FUNCTION_BLOCK FB_UAnodeReleaseHandleMock_Success IMPLEMENTS I_OPCUA_NodeReleaseHandle
VAR_INPUT
END_VAR
VAR_OUTPUT
END_VAR
VAR
END_VAR

{warning 'add method implementation '}
METHOD start : BOOL
VAR_INPUT
    Execute       : BOOL;
    ConnectionHdl : DWORD;
    NodeHdl       : DWORD;
    Timeout       : TIME := DEFAULT_ADS_TIMEOUT; 
END_VAR
VAR_OUTPUT
	Done	: BOOL;
	Busy	: BOOL;
	Error	: BOOL;
	ErrorID	: DWORD;
END_VAR
IF execute THEN
	done := TRUE;
END_IF
END_METHOD

END_FUNCTION_BLOCK

(* stored: Version 1.1.0.1, ProductVersion 3.1.4024.9
   POU FB_UAnodeReleaseHandleMock_Success: Id {88666360-9187-4fe4-99d0-ef8b00f9460c}, SpecialFunc None
   Method start: Id {0ccd4082-9455-41df-a361-fbc64e269132} *)
